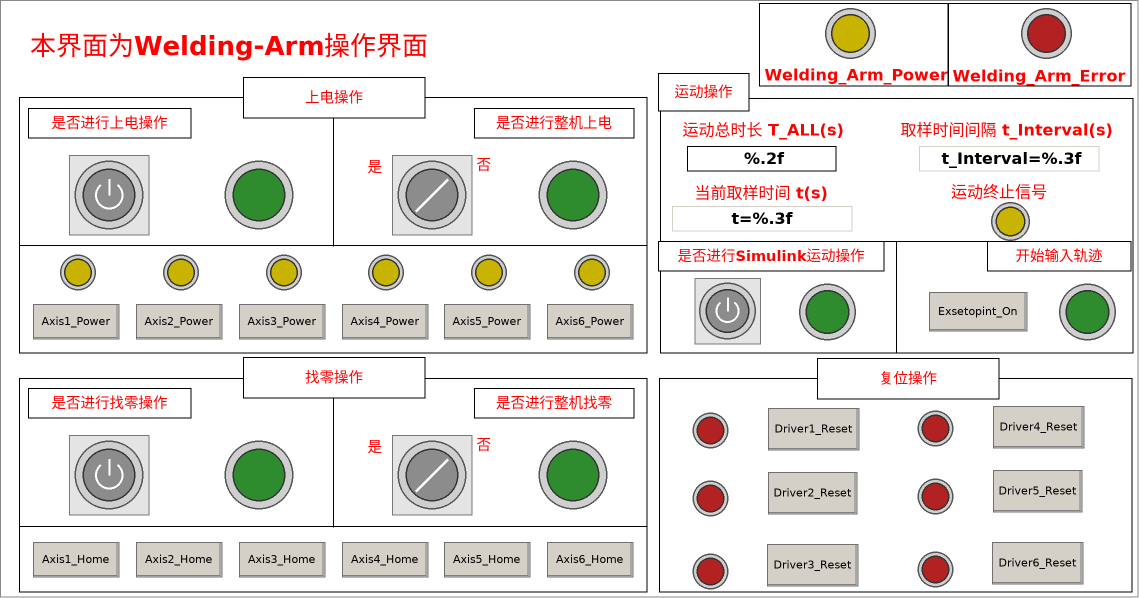
VISUALIZATION Visu_Welding_Arm_Move  // 1139x598
    Rectangle (660,98 473x255)
    Rectangle (659,378 473x214)
    Group (19,97 628x256)
        Rectangle (0,0 628x256)
        Line (1,148) (627,148)
        Line (314,0) (314,149)
    Label (345,152 60x30), "是"
    Label (454,150 60x30), "否"
    Rectangle (474,108 160x30), "是否进行整机上电"
    Lamp1 (219,155 80x80), variable: Welding_Arm_Control.Power_Execute, style: Lamp-Lamp1-Green
    Lamp1 (52,252 52x41), variable: Welding_Arm_Control.Power_Status[1], style: Lamp-Lamp1-Yellow
    Lamp1 (155,252 52x41), variable: Welding_Arm_Control.Power_Status[2], style: Lamp-Lamp1-Yellow
    Lamp1 (258,252 52x41), variable: Welding_Arm_Control.Power_Status[3], style: Lamp-Lamp1-Yellow
    Lamp1 (360,252 52x41), variable: Welding_Arm_Control.Power_Status[4], style: Lamp-Lamp1-Yellow
    Lamp1 (463,252 52x41), variable: Welding_Arm_Control.Power_Status[5], style: Lamp-Lamp1-Yellow
    Lamp1 (566,252 52x41), variable: Welding_Arm_Control.Power_Status[6], style: Lamp-Lamp1-Yellow
    Button (33,304 86x35), "Axis1_Power"
        toggle Welding_Arm_Control.Axis_Power[1]
    Button (136,304 86x35), "Axis2_Power"
        toggle Welding_Arm_Control.Axis_Power[2]
    Button (239,304 86x35), "Axis3_Power"
        toggle Welding_Arm_Control.Axis_Power[3]
    Button (342,304 86x35), "Axis4_Power"
        toggle Welding_Arm_Control.Axis_Power[4]
    Button (444,304 86x35), "Axis5_Power"
        toggle Welding_Arm_Control.Axis_Power[5]
    Button (547,304 86x35), "Axis6_Power"
        toggle Welding_Arm_Control.Axis_Power[6]
    Rectangle (28,108 163x30), "是否进行上电操作"
    PowerSwitch (69,155 80x80), variable: Welding_Arm_Control.Power_Execute, behaviour: TOGGLE, style: Switch-PowerSwitch-Gray
    Lamp1 (533,155 80x80), variable: Welding_Arm_Control.Robot_Power, style: Lamp-Lamp1-Green
    RotarySwitch (392,155 80x80), variable: Welding_Arm_Control.Welding_Arm_Power, behaviour: TOGGLE, style: Switch-RotarySwitch-Gray
    Rectangle (243,77 182x41), "上电操作"
    Group (19,378 628x214)
        Rectangle (0,0 628x214)
        Line (1,148) (627,148)
        Line (314,0) (314,149)
    Label (345,432 60x30), "是"
    Label (454,430 60x30), "否"
    Rectangle (474,388 160x30), "是否进行整机找零"
    Lamp1 (219,435 80x80), variable: Welding_Arm_Control.Power_Execute, style: Lamp-Lamp1-Green
    Button (33,542 86x35), "Axis1_Home"
        toggle Welding_Arm_Control.Axis_Home_Set[1]
    Button (136,542 86x35), "Axis2_Home"
        toggle Welding_Arm_Control.Axis_Home_Set[2]
    Button (239,542 86x35), "Axis3_Home"
        toggle Welding_Arm_Control.Axis_Home_Set[3]
    Button (342,542 86x35), "Axis4_Home"
        toggle Welding_Arm_Control.Axis_Home_Set[4]
    Button (444,542 86x35), "Axis5_Home"
        toggle Welding_Arm_Control.Axis_Home_Set[5]
    Button (547,542 86x35), "Axis6_Home"
        toggle Welding_Arm_Control.Axis_Home_Set[6]
    Rectangle (28,388 163x30), "是否进行找零操作"
    PowerSwitch (69,435 80x80), variable: Welding_Arm_Control.Home_Execute, behaviour: TOGGLE, style: Switch-PowerSwitch-Gray
    Lamp1 (533,435 80x80), variable: Welding_Arm_Control.Robot_Power, style: Lamp-Lamp1-Green
    RotarySwitch (392,435 80x80), variable: Welding_Arm_Control.Welding_Arm_Home_Set, behaviour: TOGGLE, style: Switch-RotarySwitch-Gray
    Rectangle (243,357 182x41), "找零操作"
    Rectangle (759,3 189x83)
    Rectangle (948,3 183x83)
    Lamp1 (1016,4 61x59), variable: Welding_Arm_Control.Robot_Error, style: Lamp-Lamp1-Red
    Label (953,60 172x32), "Welding_Arm_Error"
    Lamp1 (820,4 61x59), variable: Welding_Arm_Control.Robot_Power, style: Lamp-Lamp1-Yellow
    Label (766,59 181x32), "Welding_Arm_Power"
    Lamp1 (690,406 41x49), variable: Welding_Arm_Control.Axis_Error[1], style: Lamp-Lamp1-Red
    Lamp1 (690,474 41x49), variable: Welding_Arm_Control.Axis_Error[2], style: Lamp-Lamp1-Red
    Lamp1 (690,547 41x49), variable: Welding_Arm_Control.Axis_Error[3], style: Lamp-Lamp1-Red
    Button (768,408 91x42), "Driver1_Reset"
        tap Welding_Arm_Control.Axis_Reset[1]
    Button (768,472 89x42), "Driver2_Reset"
        tap Welding_Arm_Control.Axis_Reset[2]
    Button (767,544 91x42), "Driver3_Reset"
        tap Welding_Arm_Control.Axis_Reset[3]
    Lamp1 (915,404 41x49), variable: Welding_Arm_Control.Axis_Error[1], style: Lamp-Lamp1-Red
    Lamp1 (915,472 41x49), variable: Welding_Arm_Control.Axis_Error[2], style: Lamp-Lamp1-Red
    Lamp1 (915,545 41x49), variable: Welding_Arm_Control.Axis_Error[3], style: Lamp-Lamp1-Red
    Button (993,406 91x42), "Driver4_Reset"
        tap Welding_Arm_Control.Axis_Reset[4]
    Button (993,470 89x42), "Driver5_Reset"
        tap Welding_Arm_Control.Axis_Reset[5]
    Button (992,542 91x42), "Driver6_Reset"
        tap Welding_Arm_Control.Axis_Reset[6]
    Rectangle (687,146 149x25), "%.2f", text variable: Welding_Arm_Movement.T_ALL
        OnMouseClick: write Welding_Arm_Movement.T_ALL via Default
    Label (664,118 199x24), "运动总时长 T_ALL(s)"
    Textfield (672,206 180x25), "t=%.3f", text variable: Welding_Arm_Movementl.t
    Label (684,181 155x24), "当前取样时间 t(s)"
    Lamp1 (982,199 57x45), variable: Robot_Movement.ExtSetPointDisable, style: Lamp-Lamp1-Yellow
    Label (909,180 180x24), "运动终止信号"
    Label (877,118 260x24), "取样时间间隔 t_Interval(s)"
    Textfield (919,146 180x25), "t_Interval=%.3f", text variable: Welding_Arm_Movement.t_Interval
        OnMouseClick: write Welding_Arm_Movement.t_Interval via Default
    Rectangle (817,358 182x41), "复位操作"
    Line (659,241) (1131,241)
    Rectangle (658,241 226x30), "是否进行Simulink运动操作"
    Lamp1 (791,279 73x66), variable: Welding_Arm_Movement.ExSetPoint_Execute, style: Lamp-Lamp1-Green
    PowerSwitch (691,278 73x66), variable: Welding_Arm_Movement.ExSetPoint_Execute, behaviour: TOGGLE, style: Switch-PowerSwitch-Gray
    Rectangle (987,241 144x30), "开始输入轨迹"
    Button (929,292 98x39), "Exsetopint_On"
        toggle Welding_Arm_Movement.ExtSetPointEnable
    Lamp1 (1051,279 73x66), variable: Welding_Arm_Movement.ExtSetPointEnable, style: Lamp-Lamp1-Green
    Line (896,242) (896,352)
    Label (27,25 572x42), "本界面为Welding-Arm操作界面"
    Rectangle (658,73 91x38), "运动操作"
END_VISUALIZATION

(* stored: Version 1.1.0.1, ProductVersion 3.1.4020.12
   Visu Visu_Welding_Arm_Move: Id {9796b77c-13d9-45a3-9411-d28583c3b7d5} *)
